(* LS Electric XG5000 project: WEG_CFW500_FB *)
(* PLC LSPLC *)
(* module base 0 slot 0: Input/Output Module:XEM-DN/DP32HP (DC 24V Input, Transistor Output, 32 Contacts) *)
(* module base 0 slot 1: Internal Positioning:XBF-PO06E (Open Collector Type, 6 Axis) *)
(* module base 0 slot 2: EtherNet/IP:XBL-EIPT (EtherNet/IP communication module, electrical) *)
VAR_GLOBAL
    WEG_CFW500_Input00 : ARRAY[0..3] OF BYTE; (* Input data to ethernet/IP WEG CFW500 drive *)
    WEG_CFW500_Output00 : ARRAY[0..3] OF BYTE; (* Output data to ethernet/IP WEG CFW500 drive *)
END_VAR

(* Comments on direct variables
%IX0.0.0	this is comment 1
*)

TYPE WEG_CFW500_EIP_UDT : (* this is a user data type for the GS20_Drive_FB *)
STRUCT
    Status_STO : BOOL; (* Status of the drive safe torque off *)
    Status_RunCmd : BOOL; (* Status of drive run command *)
    Status_ActiveQuickStop : BOOL; (* 0: The quick stop command is not active. / 1: The drive is executing the quick stop command. *)
    Status_SecondRamp : BOOL; (* 0: The drive is configured to use the first ramp values, programmed in P0100 and P0101, as the motor / acceleration and deceleration ramp times. / 1: The drive is configured to use the second ramp values, programmed in P0102 and P0103, as the motor / acceleration and deceleration ramp times. *)
    Status_ConfigurationMode : BOOL; (* Status of configuration mode. 0: The drive is operating normally. / 1: The drive is in the configuration mode. It indicates a special condition during which the drive cannot be / enabled *)
    Status_AlarmPresent : BOOL; (* 0: The drive is not in alarm condition. / 1: The drive is in alarm condition. *)
    Status_MotorRunning : BOOL; (* 0: The motor is stopped (or coast to stop). / 1: The drive is running the motor at the set point speed, or executing either the acceleration or the deceleration / ramp. *)
    Status_ActGenEnabled : BOOL; (* 0: General Enable is not active. / 1: General Enable is active and the drive is ready to run the motor. *)
    Status_SpeedDirection : BOOL; (* 0: The motor is running in the reverse direction. / 1: The motor is running in the forward direction. *)
    Status_Jogging : BOOL; (* 0: JOG function disabled. / 1: JOG function enabled. *)
    Status_LocalRemote : BOOL; (* 0: Drive in Local mode. / 1: Drive in Remote mode. *)
    Status_Undervoltage : BOOL; (* 0: No Undervoltage. / 1: With Undervoltage. *)
    Status_ManualAuto : BOOL; (* 0: PID in manual mode. / 1: PID in Automatic mode *)
    Status_FaultPresent : BOOL; (* 0: The drive is not in a fault condition. / 1: The drive has detected a fault. *)
    Status_MotorSpeedHz : REAL; (* motor speed in Hz. *)
    Cmd_RunStop : BOOL; (* 0: It stops the motor with deceleration ramp. / 1: The motor runs according to the acceleration ramp. *)
    Cmd_GenEnable : BOOL; (* 0: It disables the drive, interrupting the supply for the motor. / 1: It enables the drive allowing the motor operation. *)
    Cmd_SpeedDirection : BOOL; (* 0: Direction of rotation is opposed to the speed reference (reverse). / 1: Direction of rotation is the same as the speed reference (direct). *)
    Cmd_Jog : BOOL; (* 0: It disables the JOG function. / 1: It enables the JOG function *)
    Cmd_LocalRemote : BOOL; (* 0: The drive goes to the Local mode. / 1: The drive goes to the Remote mode. *)
    Cmd_SecondRamp : BOOL; (* 0: The drive uses the first ramp values, programmed in P0100 and P0101, as the motor acceleration and / deceleration ramp times. / 1: The drive is configured to use the second ramp values, programmed in P0102 and P0103, as the motor / acceleration and deceleration ramp times *)
    Cmd_QuickStop : BOOL; (* 0: It does not execute the quick stop command. / 1: It executes the quick stop command. *)
    Cmd_FaultReset : BOOL; (* 0: No function. / 1: If in a fault condition, then it executes the fault reset. *)
    Cmd_SpeedReferenceHz : REAL; (* Hz speed command to drive. *)
END_STRUCT;
END_TYPE

FUNCTION_BLOCK WEG_CFW500_EIP_FB
(* This function block is used to control and receive status of a WEG CFW500 inverter drive. *)
VAR_INPUT
    Enable : BOOL; (* Enable the WEG CFW500 function block. *)
    InputData : ARRAY[0..3] OF BYTE; (* Ethernet/IP input data array from WEG CFW500 drive *)
END_VAR
VAR_IN_OUT
    WEG_CFW500_UDT : WEG_CFW500_EIP_UDT; (* User data type for WEG CFW500 *)
    OutputData : ARRAY[0..3] OF BYTE; (* Ethernet/IP output data array from WEG CFW500 drive *)
END_VAR
VAR_OUTPUT
    Active : BOOL; (* Status that WEG CFW500 function block is enabled. *)
END_VAR
VAR
    BTempInput : ARRAY[0..3] OF BYTE; (* temporary byte array *)
    BTempOutput : ARRAY[0..3] OF BYTE; (* temporary byte array *)
    ITemp : INT; (* temporary int value *)
    Temporary_Word : WORD; (* temporary word storage *)
END_VAR
(***************************************************************************************************
(* 
AutomationDirect.com has provided this code for convenience. This sample code is provided "as-is" with no expressed or implied warranty. 
 If the end user includes any of the sample code (in whole or part), it is the user's responsibility to completely modify, integrate, and test any code to ensure it meets all system and 
 safety requirements for the intended application or system.
 

	The 'WEG_CFW500_FB' function block uses data type BYTE for the InputData and OutputData.
		When creating a new module using the EDS file, select the data type WORD.
		
									Data type:: BYTE
									Input Size: 4 BYTES
									Output Size: 4 BYTES
									EDS File: eip_cfw500_v31x.eds
									
	***************************************************************************************************)
	
IF (Enable = TRUE) THEN		
	Active := TRUE;	
	
	(***********************
  	Mapping Input Data 
  	***********************)
  	
  	BTempInput :=ARY_MOVE(MOVE_NUM:=4, IN:=InputData, IN_INDX:=0, OUT_INDX:=0);	
  	
 	WEG_CFW500_UDT.Status_STO := BTempInput[0].0;
	WEG_CFW500_UDT.Status_RunCmd := BTempInput[0].1;
  	WEG_CFW500_UDT.Status_ActiveQuickStop := BTempInput[0].2;
	WEG_CFW500_UDT.Status_SecondRamp := BTempInput[0].3;
	WEG_CFW500_UDT.Status_ConfigurationMode := BTempInput[0].4;
	WEG_CFW500_UDT.Status_AlarmPresent := BTempInput[0].5;
	WEG_CFW500_UDT.Status_MotorRunning := BTempInput[0].6;
	WEG_CFW500_UDT.Status_ActGenEnabled := BTempInput[0].7;
	WEG_CFW500_UDT.Status_SpeedDirection := BTempInput[1].0;
	WEG_CFW500_UDT.Status_Jogging := BTempInput[1].1;
	WEG_CFW500_UDT.Status_LocalRemote := BTempInput[1].2;
	WEG_CFW500_UDT.Status_Undervoltage := BTempInput[1].3;
	WEG_CFW500_UDT.Status_ManualAuto := BTempInput[1].4;
	WEG_CFW500_UDT.Status_FaultPresent := BTempInput[1].5;
	
	//Status for Drive Speed in HZ
	Temporary_Word := BYTE_WORD(LOW:=BTempInput[2], HIGH:=BTempInput[3]);
	ITemp := WORD_TO_INT(IN:=Temporary_Word);
	WEG_CFW500_UDT.Status_MotorSpeedHz :=  (INT_TO_REAL(IN:=ITemp) * 60.0) / 8192.0;
	
	
	(***********************
  	Mapping Output Data 
  	***********************)
 	BTempOutput[0].0 := WEG_CFW500_UDT.Cmd_RunStop;
 	BTempOutput[0].1 := WEG_CFW500_UDT.Cmd_GenEnable;
 	BTempOutput[0].2 := WEG_CFW500_UDT.Cmd_SpeedDirection;
 	BTempOutput[0].3 := WEG_CFW500_UDT.Cmd_Jog;
 	BTempOutput[0].4 := WEG_CFW500_UDT.Cmd_LocalRemote;
 	BTempOutput[0].5 := WEG_CFW500_UDT.Cmd_SecondRamp;
 	BTempOutput[0].6 := WEG_CFW500_UDT.Cmd_QuickStop;
 	BTempOutput[0].7 := WEG_CFW500_UDT.Cmd_FaultReset;
 	
 	//CMD for Drive Speed in HZ
	ITemp :=  REAL_TO_INT((WEG_CFW500_UDT.Cmd_SpeedReferenceHz * 8192.0) / 60.0);
	Temporary_Word := INT_TO_WORD(IN:=ITemp);
 	WORD_BYTE(IN:=Temporary_Word, LOW=>BTempOutput[2], HIGH=>BTempOutput[3]);
 
 	
 	OutputData :=ARY_MOVE(MOVE_NUM:=4, IN:=BTempOutput, IN_INDX:=0, OUT_INDX:=0);


ELSE
	Active := FALSE;
END_IF;
END_FUNCTION_BLOCK

PROGRAM FB_Usage_LD (* task: Scan Program *)
VAR
    CFW500_00 : WEG_CFW500_EIP_FB; (* WEG CFW500 FB *)
    fbActive : BOOL;
    WEG_CFW500_Drive00 : WEG_CFW500_EIP_UDT; (* User data type for Weg CFW500 *)
END_VAR
VAR_EXTERNAL
    WEG_CFW500_Input00 : ARRAY[0..3] OF BYTE; (* Input data to ethernet/IP WEG CFW500 drive *)
    WEG_CFW500_Output00 : ARRAY[0..3] OF BYTE; (* Output data to ethernet/IP WEG CFW500 drive *)
END_VAR

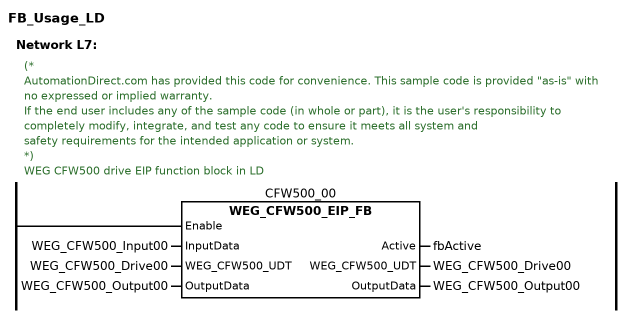
(* ( * / AutomationDirect.com has provided this code for convenience. This sample code is provided "as-is" with no expressed or implied warranty. / If the end user includes any of the sample code (in whole or part), it is the user's responsibility to completely modify, integrate, and test any code to ensure it meets all system and / safety requirements for the intended application or system. / * ) *)
(* WEG CFW500 drive EIP function block in LD *)
(* Rung L7 *)
CFW500_00(Enable := TRUE, InputData := WEG_CFW500_Input00, WEG_CFW500_UDT := WEG_CFW500_Drive00, OutputData := WEG_CFW500_Output00, Active => fbActive, WEG_CFW500_UDT => WEG_CFW500_Drive00, OutputData => WEG_CFW500_Output00);
END_PROGRAM

PROGRAM FB_Usage_ST (* task: Scan Program *)
(*  *)
VAR
    fbActive : BOOL;
    WEG_CFW500_Drive00 : WEG_CFW500_EIP_UDT; (* User data type for Weg CFW500 *)
    WEG_CFW500_FB00 : WEG_CFW500_EIP_FB; (* function block *)
END_VAR
VAR_EXTERNAL
    WEG_CFW500_Input00 : ARRAY[0..3] OF BYTE; (* Input data to ethernet/IP WEG CFW500 drive *)
    WEG_CFW500_Output00 : ARRAY[0..3] OF BYTE; (* Output data to ethernet/IP WEG CFW500 drive *)
END_VAR
(* 
AutomationDirect.com has provided this code for convenience. This sample code is provided "as-is" with no expressed or implied warranty. 
 If the end user includes any of the sample code (in whole or part), it is the user's responsibility to completely modify, integrate, and test any code to ensure it meets all system and 
 safety requirements for the intended application or system.
 *)





WEG_CFW500_FB00(Enable:=TRUE, InputData:=WEG_CFW500_Input00, WEG_CFW500_UDT:=WEG_CFW500_Drive00, OutputData:=WEG_CFW500_Output00, Active=>fbActive);
END_PROGRAM